PROGRAM AddCommand
VAR
END_VAR

IF GVL_MOTION.EXT_CTR.CMDADD THEN
	GVL_MOTION.EXT_CTR.CMDADD					:= FALSE;
	//QueueEnd contains no data
	IF GVL_MOTION.ScriptEnd < 100 THEN
		GVL_MOTION.Script[GVL_MOTION.ScriptEnd]	:= GVL_MOTION.InstructionBuffer;
		GVL_MOTION.ScriptEnd 					:= GVL_MOTION.ScriptEnd + 1;
		GVL_MOTION.EXT_CTR.CMDADD 				:= FALSE;
	ELSE
		//error msg
		GVL_MOTION.EXT_CTR.CMDADD 				:= FALSE;
	END_IF

END_IF

END_PROGRAM

(* stored: Version 1.1.0.1, ProductVersion 3.1.4026.18
   POU AddCommand: Id {9bb5efea-5d4b-4d82-83e6-06192cbb2d4f}, SpecialFunc None *)
